// TIA Portal project "Ascensor" (V14)

(* hardware
DEVICE "S7-1200 station_1"  S7-1200 Station
   slot 0: "Rack_0"  S7-1200 Rack  Rack  V1.0
   slot 1: "PLC_1"  CPU 1214C AC/DC/Rly  6ES7 214-1BG40-0XB0  V4.0
*)

// ===== PLC "PLC_1"  CPU 1214C AC/DC/Rly =====

VAR_GLOBAL   // PLC tag table "Estados"
   "0" AT %M10.0 : Bool;   // Marcha/Paro del sistema
   "1" AT %M10.1 : Bool;   // Marcha/Paro del sistema
   "2" AT %M10.2 : Bool;   // Marcha/Paro del sistema
   "10" AT %M10.3 : Bool;   // Selección modo
   "11" AT %M10.4 : Bool;   // Selección modo
   "12" AT %M10.5 : Bool;   // Selección modo
   "20" AT %M10.6 : Bool;   // Movimiento de la cabina
   "21" AT %M10.7 : Bool;   // Movimiento de la cabina
   "22" AT %M11.0 : Bool;   // Movimiento de la cabina
   "23" AT %M11.1 : Bool;   // Movimiento de la cabina
   "24" AT %M11.2 : Bool;   // Movimiento de la cabina
   "25" AT %M11.3 : Bool;   // Movimiento de la cabina
   "30" AT %M11.4 : Bool;   // Apertura y Cierre de Puerta
   "31" AT %M11.5 : Bool;   // Apertura y Cierre de Puerta
   "32" AT %M11.6 : Bool;   // Apertura y Cierre de Puerta
   "33" AT %M11.7 : Bool;   // Apertura y Cierre de Puerta
   "34" AT %M12.0 : Bool;   // Apertura y Cierre de Puerta
   "35" AT %M12.1 : Bool;   // Apertura y Cierre de Puerta
   "40" AT %M12.2 : Bool;   // Reset llamda y memoria
   "41" AT %M12.3 : Bool;   // Reset llamda y memoria
   "42" AT %M12.4 : Bool;   // Reset llamda y memoria
   "43" AT %M12.5 : Bool;   // Reset llamda y memoria
   "50" AT %M12.6 : Bool;   // Órdenes automáticas de subida y bajada
   "51" AT %M12.7 : Bool;   // Órdenes automáticas de subida y bajada
   "52" AT %M13.0 : Bool;   // Órdenes automáticas de subida y bajada
   "60" AT %M13.1 : Bool;   // Órdenes manuales de subida y bajada
   "61" AT %M13.2 : Bool;   // Órdenes manuales de subida y bajada
   "62" AT %M13.3 : Bool;   // Órdenes manuales de subida y bajada
   "63" AT %M13.4 : Bool;   // Órdenes manuales de subida y bajada
   "64" AT %M13.5 : Bool;   // Órdenes manuales de subida y bajada
   "65" AT %M13.6 : Bool;   // Órdenes manuales de subida y bajada
   "66" AT %M13.7 : Bool;   // Órdenes manuales de subida y bajada
   "70" AT %M14.0 : Bool;   // Detección de errores
   "71" AT %M14.1 : Bool;   // Detección de errores
   "72" AT %M14.2 : Bool;   // Detección de errores
   "73" AT %M14.3 : Bool;   // Detección de errores
   "74" AT %M14.4 : Bool;   // Detección de errores
   "75" AT %M14.5 : Bool;   // Detección de errores
   "80" AT %M14.6 : Bool;   // Gestión de errores
   "81" AT %M14.7 : Bool;   // Gestión de errores
   "82" AT %M15.0 : Bool;   // Gestión de errores
   "83" AT %M15.1 : Bool;   // Gestión de errores
   "84" AT %M15.2 : Bool;   // Gestión de errores
   "85" AT %M15.3 : Bool;   // Gestión de errores
   "86" AT %M15.4 : Bool;   // Gestión de errores
   "87" AT %M15.5 : Bool;   // Gestión de errores
   "88" AT %M15.6 : Bool;   // Gestión de errores
   "90" AT %M15.7 : Bool;   // Descenso a primera planta
   "91" AT %M16.0 : Bool;   // Descenso a primera planta
   "92" AT %M16.1 : Bool;   // Descenso a primera planta
END_VAR

VAR_GLOBAL   // PLC tag table "Salidas"
   "LBC0" AT %M30.0 : Bool;   // Lámpara Pulsador Cabina Planta 0
   "LBC1" AT %M30.1 : Bool;   // Lámpara Pulsador Cabina Planta 1
   "LBC2" AT %M30.2 : Bool;   // Lámpara Pulsador Cabina Planta 2
   "LBC3" AT %M30.3 : Bool;   // Lámpara Pulsador Cabina Planta 3
   "LBP0" AT %M30.4 : Bool;   // Lámpara Pulsador Planta 0
   "LBP1" AT %M30.5 : Bool;   // Lámpara Pulsador Planta 1
   "LBP2" AT %M30.6 : Bool;   // Lámpara Pulsador Planta 2
   "LBP3" AT %M30.7 : Bool;   // Lámpara Pulsador Planta 3
   "MCD" AT %M31.0 : Bool;   // Orden Giro Motor Cabina Derecha - Ascender
   "MCI" AT %M31.1 : Bool;   // Orden Giro Motor Cabina Izquierda - Descender
   "MPD" AT %M31.2 : Bool;   // Orden Giro Motor Puerta Derecha - Apertura
   "MPI" AT %M31.3 : Bool;   // Orden Giro Motor Puerta Izquierda - Cierre
   "LA" AT %M31.4 : Bool;   // Lámpara Indicadora Llamada Ascendente
   "LD" AT %M31.5 : Bool;   // Lámpara Indicadora Llamada Descendente
   "Z" AT %M31.6 : Bool;   // Zumbador Indicador de Llamada
END_VAR

VAR_GLOBAL   // PLC tag table "Variables Internas"
   "Pos0" AT %M20.0 : Bool;   // Cabina en Planta 0
   "Pos1" AT %M20.1 : Bool;   // Cabina en Planta 1
   "Pos2" AT %M20.2 : Bool;   // Cabina en Planta 2
   "Pos3" AT %M20.3 : Bool;   // Cabina en Planta 3
   "Call0" AT %M20.4 : Bool;   // Llamada en Planta 0
   "Call1" AT %M20.5 : Bool;   // Llamada en Planta 1
   "Call2" AT %M20.6 : Bool;   // Llamada en Planta 2
   "Call3" AT %M20.7 : Bool;   // Llamada en Planta 3
   "hayCall" AT %M21.0 : Bool;   // Existencia Llamadas Pendietnes
   "upCall" AT %M21.1 : Bool;   // Llamada Ascender
   "downCall" AT %M21.2 : Bool;   // Llamada Descender
   "call_currentFloor" AT %M21.3 : Bool;   // Posición Cabina coincide con llamada
   "resetCall" AT %M21.4 : Bool;   // Finalizar llamda respondida
   "memUp" AT %M21.5 : Bool;   // Memoria Cabina Ascendiendo
   "memDown" AT %M21.6 : Bool;   // Memoria Cabina Descendiendo
   "sistemaActivado" AT %M21.7 : Bool;   // Estado General del Sistema
   "descenderPrimeraPlanta" AT %M22.0 : Bool;   // Descender a la primera planta
   "modoManual" AT %M22.1 : Bool;   // Activación del modo manual
   "modoAuto" AT %M22.2 : Bool;   // Activación del modo automático
   "abrirPuertas" AT %M22.3 : Bool;   // Iniciar secuencia de apertura de puertas
   "esperandoOrden" AT %M22.4 : Bool;   // Iniciar secuencia de decisión sobre el movimiento
   "error1" AT %M22.5 : Bool;   // Indicador de emergencia tipo 1
   "error2" AT %M22.6 : Bool;   // Indicador de emergencia tipo 2
   "modoSeguridad" AT %M22.7 : Bool;   // Indicador del estado del sistema
   "moveUp" AT %M23.0 : Bool;   // Orden de ascender
   "moveDown" AT %M23.1 : Bool;   // Orden de descender
   "finalizaLlamada" AT %M23.2 : Bool;   // Resetea una llamada
   "deleteAllCalls" AT %M23.3 : Bool;   // Resetea todas las llamadas
END_VAR

VAR_GLOBAL   // PLC tag table "Entradas"
   "BC0" AT %M0.0 : Bool;   // Pulsador Cabina Planta 0
   "BC1" AT %M0.1 : Bool;   // Pulsador Cabina Planta 1
   "BC2" AT %M0.2 : Bool;   // Pulsador Cabina Planta 2
   "BC3" AT %M0.3 : Bool;   // Pulsador Cabina Planta 3
   "BCC" AT %M0.4 : Bool;   // Pulsador Cabina Cierre Puertas
   "BCA" AT %M0.5 : Bool;   // Pulsador Cabina Apertura Puertas
   "BP0" AT %M0.6 : Bool;   // Pulsador Planta 0
   "BP1" AT %M0.7 : Bool;   // Pulsador Planta 1
   "BP2" AT %M1.0 : Bool;   // Pulsador Planta 2
   "BP3" AT %M1.1 : Bool;   // Pulsador Planta 3
   "IBL0" AT %M1.2 : Bool;   // Interruptor Biestable Lengüeta Planta 0
   "IBL1" AT %M1.3 : Bool;   // Interruptor Biestable Lengüeta Planta 1
   "IBL2" AT %M1.4 : Bool;   // Interruptor Biestable Lengüeta Planta 2
   "IBL3" AT %M1.5 : Bool;   // Interruptor Biestable Lengüeta Planta 3
   "FCPA" AT %M1.6 : Bool;   // Final de Carrera Puerta Apertura
   "FCPC" AT %M1.7 : Bool;   // Final de Carrera Puerta Cierre
   "SO" AT %M2.0 : Bool;   // Sensor Obstáculo Puerta Cabina
   "SC" AT %M2.1 : Bool;   // Sensor Carga Cabina
   "Activar" AT %M2.2 : Bool;   // Señal de Activación del sistema
   "Desactivar" AT %M2.3 : Bool;   // Señal de Desactivación del sistema
   "MA" AT %M2.4 : Bool;   // Señal de selección del modo manual
   "AUTO" AT %M2.5 : Bool;   // Señal de selección del modo automático
   "emergenciaParada" AT %M2.6 : Bool;   // Señal de emergencia que requiere parada
   "finEmergenciaParada" AT %M2.7 : Bool;   // Señal fin de emergencia que requiere parada
   "emergenciaPrimeraPlanta" AT %M3.0 : Bool;   // Señal de emergencia que requiere descender a la primera planta
   "finEmergenciaPrimeraPlanta" AT %M3.1 : Bool;   // Señal de fin de emergencia que requiere descender a primera planta
   "BA" AT %M3.2 : Bool;   // Botón Ascender Manual
   "BD" AT %M3.3 : Bool;   // Botón Descender Manual
   "BI" AT %M3.4 : Bool;   // Botón Ignorar Manual
END_VAR

// folder: System blocks/Program resources

DATA_BLOCK "TimerPuertas"   // DB3
{ S7_Optimized_Access := 'TRUE' }
AUTHOR : Simatic
FAMILY : IEC
NAME : IEC_TMR
VERSION : 1.0
// stored: InstanceOfName IEC_TIMER
"IEC_TIMER"
BEGIN
END_DATA_BLOCK

// folder: (top level)

ORGANIZATION_BLOCK "Main"   // OB1, LAD, ProgramCycle
TITLE = "Main Program Sweep (Cycle)"
{ S7_Optimized_Access := 'TRUE' }
VERSION : 0.1
   VAR_INPUT
      Initial_Call : Bool;   // Initial call of this OB
      Remanence : Bool;   // =True, if remanent data are available
   END_VAR
   VAR_TEMP   // added for the SCL form of the ladder/FBD networks
      _w1 : Bool;
      _w2 : Bool;
      _w3 : Bool;
   END_VAR
BEGIN

REGION Network 1: Variables Internas Posición Cabina
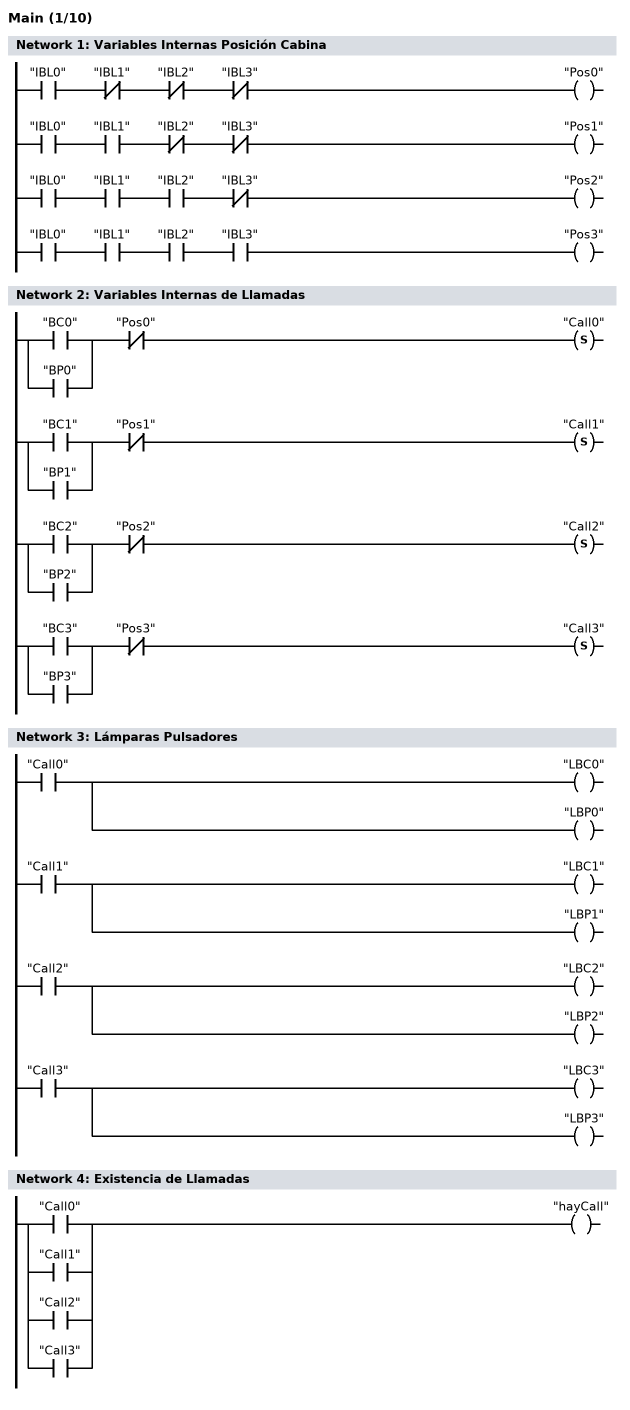
   RUNG wire#powerrail
      Contact( "IBL0" )
      I_Contact( "IBL1" )
      I_Contact( "IBL2" )
      I_Contact( "IBL3" )
      Coil( "Pos0" )
   END_RUNG
   RUNG wire#powerrail
      Contact( "IBL0" )
      Contact( "IBL1" )
      I_Contact( "IBL2" )
      I_Contact( "IBL3" )
      Coil( "Pos1" )
   END_RUNG
   RUNG wire#powerrail
      Contact( "IBL0" )
      Contact( "IBL1" )
      Contact( "IBL2" )
      I_Contact( "IBL3" )
      Coil( "Pos2" )
   END_RUNG
   RUNG wire#powerrail
      Contact( "IBL0" )
      Contact( "IBL1" )
      Contact( "IBL2" )
      Contact( "IBL3" )
      Coil( "Pos3" )
   END_RUNG
   // the same network as SCL:
   "Pos0" := "IBL0" AND NOT "IBL1" AND NOT "IBL2" AND NOT "IBL3";
   "Pos1" := "IBL0" AND "IBL1" AND NOT "IBL2" AND NOT "IBL3";
   "Pos2" := "IBL0" AND "IBL1" AND "IBL2" AND NOT "IBL3";
   "Pos3" := "IBL0" AND "IBL1" AND "IBL2" AND "IBL3";
END_REGION

REGION Network 2: Variables Internas de Llamadas
   RUNG wire#powerrail
      Contact( "BC0" )
      wire#w1
      I_Contact( "Pos0" )
      S_Coil( "Call0" )
   END_RUNG
   RUNG wire#powerrail
      Contact( "BP0" )
   END_RUNG wire#w1
   RUNG wire#powerrail
      Contact( "BC1" )
      wire#w2
      I_Contact( "Pos1" )
      S_Coil( "Call1" )
   END_RUNG
   RUNG wire#powerrail
      Contact( "BP1" )
   END_RUNG wire#w2
   RUNG wire#powerrail
      Contact( "BC2" )
      wire#w3
      I_Contact( "Pos2" )
      S_Coil( "Call2" )
   END_RUNG
   RUNG wire#powerrail
      Contact( "BP2" )
   END_RUNG wire#w3
   RUNG wire#powerrail
      Contact( "BC3" )
      wire#w4
      I_Contact( "Pos3" )
      S_Coil( "Call3" )
   END_RUNG
   RUNG wire#powerrail
      Contact( "BP3" )
   END_RUNG wire#w4
   // the same network as SCL:
   IF ("BC0" OR "BP0") AND NOT "Pos0" THEN "Call0" := TRUE; END_IF;
   IF ("BC1" OR "BP1") AND NOT "Pos1" THEN "Call1" := TRUE; END_IF;
   IF ("BC2" OR "BP2") AND NOT "Pos2" THEN "Call2" := TRUE; END_IF;
   IF ("BC3" OR "BP3") AND NOT "Pos3" THEN "Call3" := TRUE; END_IF;
END_REGION

REGION Network 3: Lámparas Pulsadores
   RUNG wire#powerrail
      Contact( "Call0" )
      wire#w1
      Coil( "LBC0" )
   END_RUNG
   RUNG wire#w1
      Coil( "LBP0" )
   END_RUNG
   RUNG wire#powerrail
      Contact( "Call1" )
      wire#w2
      Coil( "LBC1" )
   END_RUNG
   RUNG wire#w2
      Coil( "LBP1" )
   END_RUNG
   RUNG wire#powerrail
      Contact( "Call2" )
      wire#w3
      Coil( "LBC2" )
   END_RUNG
   RUNG wire#w3
      Coil( "LBP2" )
   END_RUNG
   RUNG wire#powerrail
      Contact( "Call3" )
      wire#w4
      Coil( "LBC3" )
   END_RUNG
   RUNG wire#w4
      Coil( "LBP3" )
   END_RUNG
   // the same network as SCL:
   "LBC0" := "Call0";
   "LBP0" := "Call0";
   "LBC1" := "Call1";
   "LBP1" := "Call1";
   "LBC2" := "Call2";
   "LBP2" := "Call2";
   "LBC3" := "Call3";
   "LBP3" := "Call3";
END_REGION

REGION Network 4: Existencia de Llamadas
   RUNG wire#powerrail
      Contact( "Call0" )
      wire#w1
      Coil( "hayCall" )
   END_RUNG
   RUNG wire#powerrail
      Contact( "Call1" )
   END_RUNG wire#w1
   RUNG wire#powerrail
      Contact( "Call2" )
   END_RUNG wire#w1
   RUNG wire#powerrail
      Contact( "Call3" )
   END_RUNG wire#w1
   // the same network as SCL:
   "hayCall" := "Call0" OR "Call1" OR "Call2" OR "Call3";
END_REGION

REGION Network 5: Dirección de las llamadas
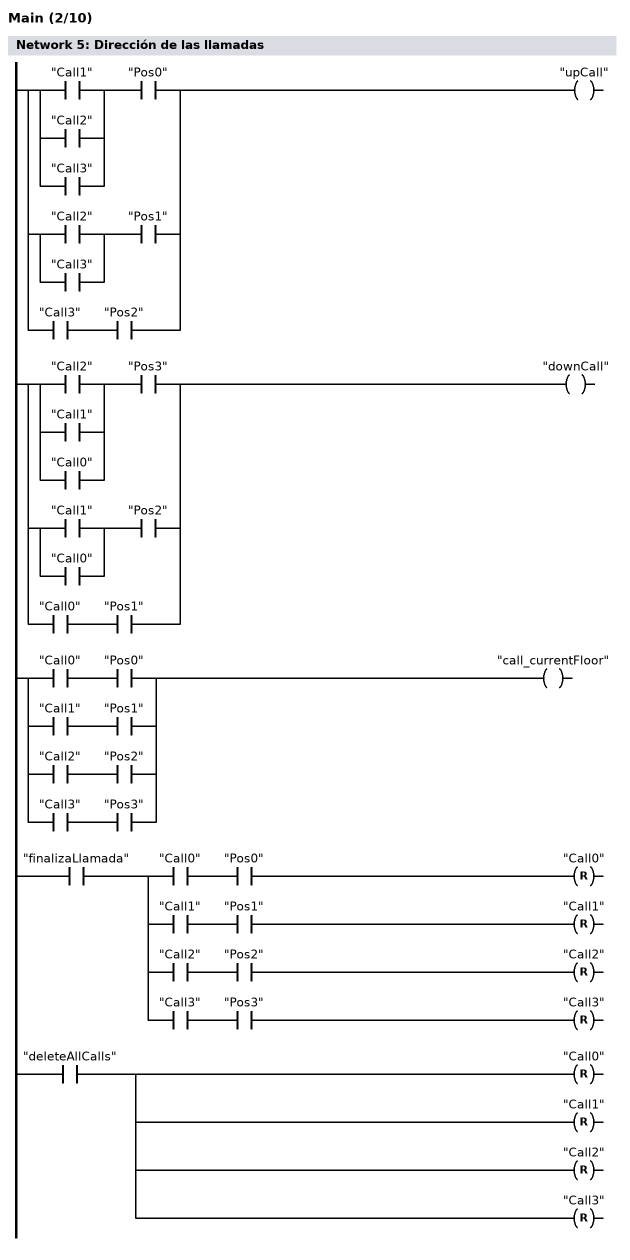
   RUNG wire#powerrail
      Contact( "Call1" )
      wire#w1
      Contact( "Pos0" )
      wire#w2
      Coil( "upCall" )
   END_RUNG
   RUNG wire#powerrail
      Contact( "Call2" )
   END_RUNG wire#w1
   RUNG wire#powerrail
      Contact( "Call3" )
   END_RUNG wire#w1
   RUNG wire#powerrail
      Contact( "Call2" )
      wire#w3
      Contact( "Pos1" )
   END_RUNG wire#w2
   RUNG wire#powerrail
      Contact( "Call3" )
   END_RUNG wire#w3
   RUNG wire#powerrail
      Contact( "Call3" )
      Contact( "Pos2" )
   END_RUNG wire#w2
   RUNG wire#powerrail
      Contact( "Call2" )
      wire#w4
      Contact( "Pos3" )
      wire#w5
      Coil( "downCall" )
   END_RUNG
   RUNG wire#powerrail
      Contact( "Call1" )
   END_RUNG wire#w4
   RUNG wire#powerrail
      Contact( "Call0" )
   END_RUNG wire#w4
   RUNG wire#powerrail
      Contact( "Call1" )
      wire#w6
      Contact( "Pos2" )
   END_RUNG wire#w5
   RUNG wire#powerrail
      Contact( "Call0" )
   END_RUNG wire#w6
   RUNG wire#powerrail
      Contact( "Call0" )
      Contact( "Pos1" )
   END_RUNG wire#w5
   RUNG wire#powerrail
      Contact( "Call0" )
      Contact( "Pos0" )
      wire#w7
      Coil( "call_currentFloor" )
   END_RUNG
   RUNG wire#powerrail
      Contact( "Call1" )
      Contact( "Pos1" )
   END_RUNG wire#w7
   RUNG wire#powerrail
      Contact( "Call2" )
      Contact( "Pos2" )
   END_RUNG wire#w7
   RUNG wire#powerrail
      Contact( "Call3" )
      Contact( "Pos3" )
   END_RUNG wire#w7
   RUNG wire#powerrail
      Contact( "finalizaLlamada" )
      wire#w8
      Contact( "Call0" )
      Contact( "Pos0" )
      R_Coil( "Call0" )
   END_RUNG
   RUNG wire#w8
      Contact( "Call1" )
      Contact( "Pos1" )
      R_Coil( "Call1" )
   END_RUNG
   RUNG wire#w8
      Contact( "Call2" )
      Contact( "Pos2" )
      R_Coil( "Call2" )
   END_RUNG
   RUNG wire#w8
      Contact( "Call3" )
      Contact( "Pos3" )
      R_Coil( "Call3" )
   END_RUNG
   RUNG wire#powerrail
      Contact( "deleteAllCalls" )
      wire#w9
      R_Coil( "Call0" )
   END_RUNG
   RUNG wire#w9
      R_Coil( "Call1" )
   END_RUNG
   RUNG wire#w9
      R_Coil( "Call2" )
   END_RUNG
   RUNG wire#w9
      R_Coil( "Call3" )
   END_RUNG
   // the same network as SCL:
   "upCall" := (("Call1" OR "Call2" OR "Call3") AND "Pos0") OR (("Call2" OR "Call3") AND "Pos1") OR ("Call3" AND "Pos2");
   "downCall" := (("Call2" OR "Call1" OR "Call0") AND "Pos3") OR (("Call1" OR "Call0") AND "Pos2") OR ("Call0" AND "Pos1");
   "call_currentFloor" := ("Call0" AND "Pos0") OR ("Call1" AND "Pos1") OR ("Call2" AND "Pos2") OR ("Call3" AND "Pos3");
   IF "finalizaLlamada" AND "Call0" AND "Pos0" THEN "Call0" := FALSE; END_IF;
   IF "finalizaLlamada" AND "Call1" AND "Pos1" THEN "Call1" := FALSE; END_IF;
   IF "finalizaLlamada" AND "Call2" AND "Pos2" THEN "Call2" := FALSE; END_IF;
   IF "finalizaLlamada" AND "Call3" AND "Pos3" THEN "Call3" := FALSE; END_IF;
   IF "deleteAllCalls" THEN
       "Call0" := FALSE;
       "Call1" := FALSE;
       "Call2" := FALSE;
       "Call3" := FALSE;
   END_IF;
END_REGION

REGION Network 6: Marcha/Paro del sistema
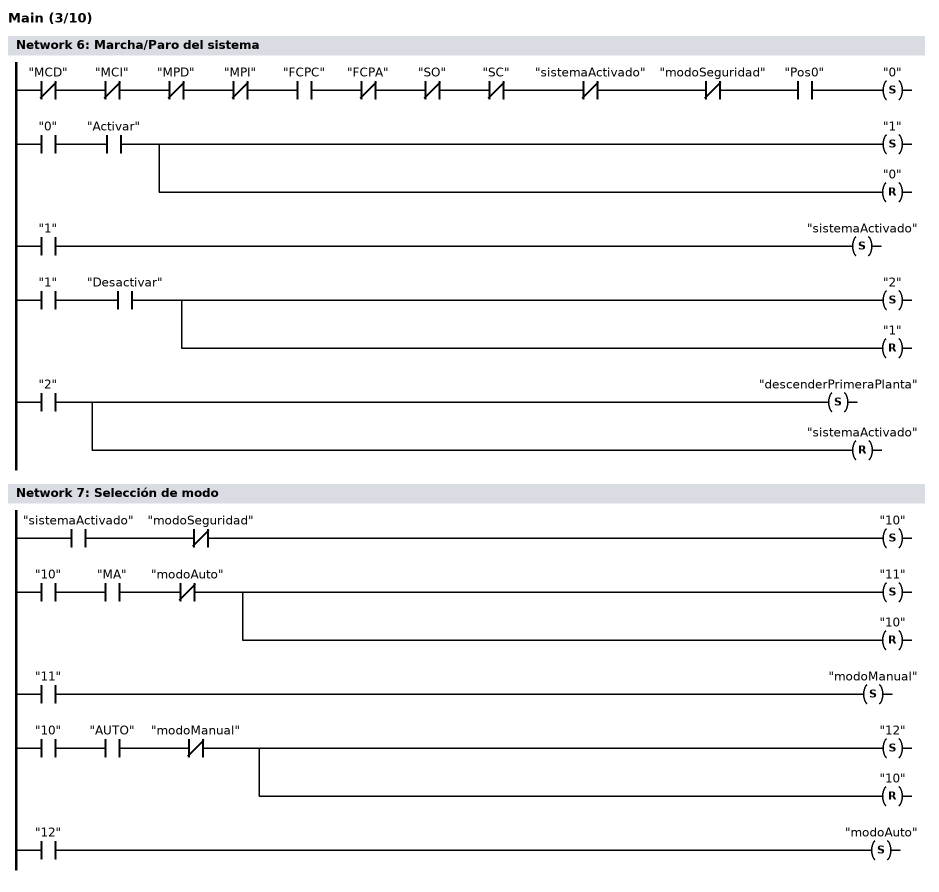
   RUNG wire#powerrail
      I_Contact( "MCD" )
      I_Contact( "MCI" )
      I_Contact( "MPD" )
      I_Contact( "MPI" )
      Contact( "FCPC" )
      I_Contact( "FCPA" )
      I_Contact( "SO" )
      I_Contact( "SC" )
      I_Contact( "sistemaActivado" )
      I_Contact( "modoSeguridad" )
      Contact( "Pos0" )
      S_Coil( "0" )
   END_RUNG
   RUNG wire#powerrail
      Contact( "0" )
      Contact( "Activar" )
      wire#w1
      S_Coil( "1" )
   END_RUNG
   RUNG wire#w1
      R_Coil( "0" )
   END_RUNG
   RUNG wire#powerrail
      Contact( "1" )
      S_Coil( "sistemaActivado" )
   END_RUNG
   RUNG wire#powerrail
      Contact( "1" )
      Contact( "Desactivar" )
      wire#w2
      S_Coil( "2" )
   END_RUNG
   RUNG wire#w2
      R_Coil( "1" )
   END_RUNG
   RUNG wire#powerrail
      Contact( "2" )
      wire#w3
      S_Coil( "descenderPrimeraPlanta" )
   END_RUNG
   RUNG wire#w3
      R_Coil( "sistemaActivado" )
   END_RUNG
   // the same network as SCL:
   IF NOT "MCD" AND NOT "MCI" AND NOT "MPD" AND NOT "MPI" AND "FCPC" AND NOT "FCPA" AND NOT "SO" AND NOT "SC" AND NOT "sistemaActivado" AND NOT "modoSeguridad" AND "Pos0" THEN
       "0" := TRUE;
   END_IF;
   IF "0" AND "Activar" THEN
       "1" := TRUE;
       "0" := FALSE;
   END_IF;
   IF "1" THEN "sistemaActivado" := TRUE; END_IF;
   IF "1" AND "Desactivar" THEN
       "2" := TRUE;
       "1" := FALSE;
   END_IF;
   IF "2" THEN
       "descenderPrimeraPlanta" := TRUE;
       "sistemaActivado" := FALSE;
   END_IF;
END_REGION

REGION Network 7: Selección de modo
   RUNG wire#powerrail
      Contact( "sistemaActivado" )
      I_Contact( "modoSeguridad" )
      S_Coil( "10" )
   END_RUNG
   RUNG wire#powerrail
      Contact( "10" )
      Contact( "MA" )
      I_Contact( "modoAuto" )
      wire#w1
      S_Coil( "11" )
   END_RUNG
   RUNG wire#w1
      R_Coil( "10" )
   END_RUNG
   RUNG wire#powerrail
      Contact( "11" )
      S_Coil( "modoManual" )
   END_RUNG
   RUNG wire#powerrail
      Contact( "10" )
      Contact( "AUTO" )
      I_Contact( "modoManual" )
      wire#w2
      S_Coil( "12" )
   END_RUNG
   RUNG wire#w2
      R_Coil( "10" )
   END_RUNG
   RUNG wire#powerrail
      Contact( "12" )
      S_Coil( "modoAuto" )
   END_RUNG
   // the same network as SCL:
   IF "sistemaActivado" AND NOT "modoSeguridad" THEN "10" := TRUE; END_IF;
   IF "10" AND "MA" AND NOT "modoAuto" THEN
       "11" := TRUE;
       "10" := FALSE;
   END_IF;
   IF "11" THEN "modoManual" := TRUE; END_IF;
   IF "10" AND "AUTO" AND NOT "modoManual" THEN
       "12" := TRUE;
       "10" := FALSE;
   END_IF;
   IF "12" THEN "modoAuto" := TRUE; END_IF;
END_REGION

REGION Network 8: Movimiento de la cabina
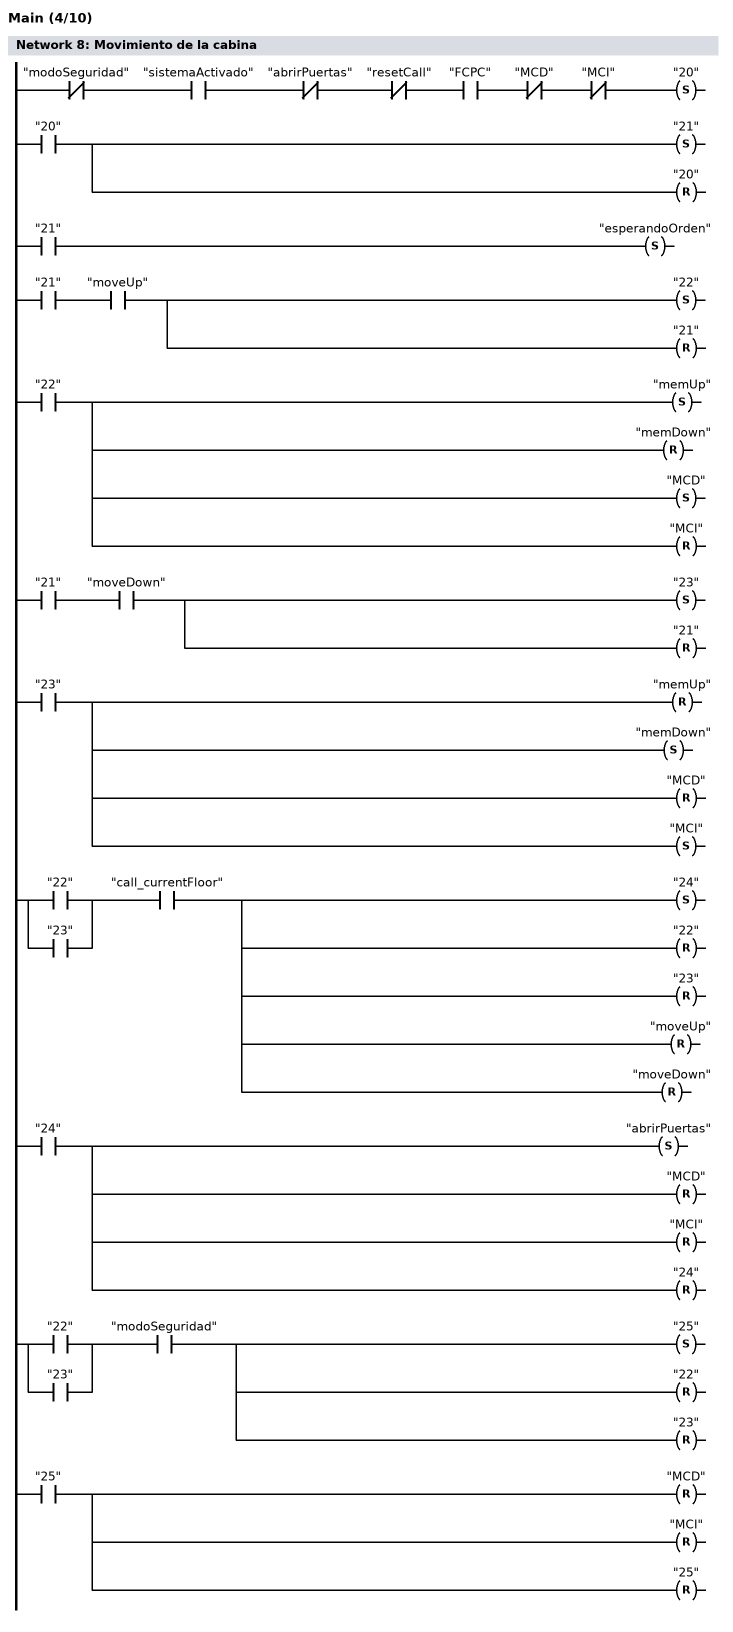
   RUNG wire#powerrail
      I_Contact( "modoSeguridad" )
      Contact( "sistemaActivado" )
      I_Contact( "abrirPuertas" )
      I_Contact( "resetCall" )
      Contact( "FCPC" )
      I_Contact( "MCD" )
      I_Contact( "MCI" )
      S_Coil( "20" )
   END_RUNG
   RUNG wire#powerrail
      Contact( "20" )
      wire#w1
      S_Coil( "21" )
   END_RUNG
   RUNG wire#w1
      R_Coil( "20" )
   END_RUNG
   RUNG wire#powerrail
      Contact( "21" )
      S_Coil( "esperandoOrden" )
   END_RUNG
   RUNG wire#powerrail
      Contact( "21" )
      Contact( "moveUp" )
      wire#w2
      S_Coil( "22" )
   END_RUNG
   RUNG wire#w2
      R_Coil( "21" )
   END_RUNG
   RUNG wire#powerrail
      Contact( "22" )
      wire#w3
      S_Coil( "memUp" )
   END_RUNG
   RUNG wire#w3
      R_Coil( "memDown" )
   END_RUNG
   RUNG wire#w3
      S_Coil( "MCD" )
   END_RUNG
   RUNG wire#w3
      R_Coil( "MCI" )
   END_RUNG
   RUNG wire#powerrail
      Contact( "21" )
      Contact( "moveDown" )
      wire#w4
      S_Coil( "23" )
   END_RUNG
   RUNG wire#w4
      R_Coil( "21" )
   END_RUNG
   RUNG wire#powerrail
      Contact( "23" )
      wire#w5
      R_Coil( "memUp" )
   END_RUNG
   RUNG wire#w5
      S_Coil( "memDown" )
   END_RUNG
   RUNG wire#w5
      R_Coil( "MCD" )
   END_RUNG
   RUNG wire#w5
      S_Coil( "MCI" )
   END_RUNG
   RUNG wire#powerrail
      Contact( "22" )
      wire#w6
      Contact( "call_currentFloor" )
      wire#w7
      S_Coil( "24" )
   END_RUNG
   RUNG wire#powerrail
      Contact( "23" )
   END_RUNG wire#w6
   RUNG wire#w7
      R_Coil( "22" )
   END_RUNG
   RUNG wire#w7
      R_Coil( "23" )
   END_RUNG
   RUNG wire#w7
      R_Coil( "moveUp" )
   END_RUNG
   RUNG wire#w7
      R_Coil( "moveDown" )
   END_RUNG
   RUNG wire#powerrail
      Contact( "24" )
      wire#w8
      S_Coil( "abrirPuertas" )
   END_RUNG
   RUNG wire#w8
      R_Coil( "MCD" )
   END_RUNG
   RUNG wire#w8
      R_Coil( "MCI" )
   END_RUNG
   RUNG wire#w8
      R_Coil( "24" )
   END_RUNG
   RUNG wire#powerrail
      Contact( "22" )
      wire#w9
      Contact( "modoSeguridad" )
      wire#w10
      S_Coil( "25" )
   END_RUNG
   RUNG wire#powerrail
      Contact( "23" )
   END_RUNG wire#w9
   RUNG wire#w10
      R_Coil( "22" )
   END_RUNG
   RUNG wire#w10
      R_Coil( "23" )
   END_RUNG
   RUNG wire#powerrail
      Contact( "25" )
      wire#w11
      R_Coil( "MCD" )
   END_RUNG
   RUNG wire#w11
      R_Coil( "MCI" )
   END_RUNG
   RUNG wire#w11
      R_Coil( "25" )
   END_RUNG
   // the same network as SCL:
   IF NOT "modoSeguridad" AND "sistemaActivado" AND NOT "abrirPuertas" AND NOT "resetCall" AND "FCPC" AND NOT "MCD" AND NOT "MCI" THEN
       "20" := TRUE;
   END_IF;
   IF "20" THEN
       "21" := TRUE;
       "20" := FALSE;
   END_IF;
   IF "21" THEN "esperandoOrden" := TRUE; END_IF;
   IF "21" AND "moveUp" THEN
       "22" := TRUE;
       "21" := FALSE;
   END_IF;
   IF "22" THEN
       "memUp" := TRUE;
       "memDown" := FALSE;
       "MCD" := TRUE;
       "MCI" := FALSE;
   END_IF;
   IF "21" AND "moveDown" THEN
       "23" := TRUE;
       "21" := FALSE;
   END_IF;
   IF "23" THEN
       "memUp" := FALSE;
       "memDown" := TRUE;
       "MCD" := FALSE;
       "MCI" := TRUE;
   END_IF;
   IF ("22" OR "23") AND "call_currentFloor" THEN "24" := TRUE; END_IF;
   #_w1 := ("22" OR "23") AND "call_currentFloor";
   IF #_w1 THEN
       "22" := FALSE;
       "23" := FALSE;
       "moveUp" := FALSE;
       "moveDown" := FALSE;
   END_IF;
   IF "24" THEN
       "abrirPuertas" := TRUE;
       "MCD" := FALSE;
       "MCI" := FALSE;
       "24" := FALSE;
   END_IF;
   IF ("22" OR "23") AND "modoSeguridad" THEN "25" := TRUE; END_IF;
   #_w2 := ("22" OR "23") AND "modoSeguridad";
   IF #_w2 THEN
       "22" := FALSE;
       "23" := FALSE;
   END_IF;
   IF "25" THEN
       "MCD" := FALSE;
       "MCI" := FALSE;
       "25" := FALSE;
   END_IF;
END_REGION

REGION Network 9: Apertura y cierre de puertas
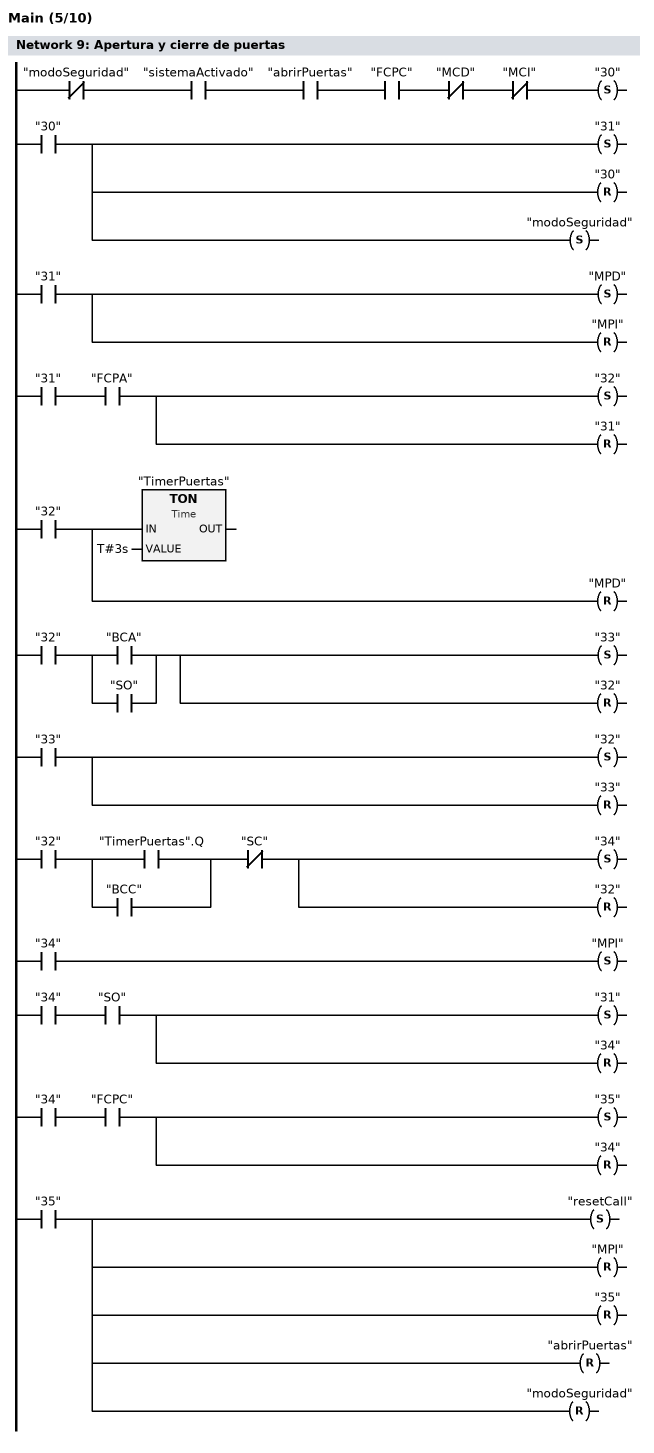
   IF NOT "modoSeguridad" AND "sistemaActivado" AND "abrirPuertas" AND "FCPC" AND NOT "MCD" AND NOT "MCI" THEN
       "30" := TRUE;
   END_IF;
   IF "30" THEN "31" := TRUE; END_IF;
   #_w1 := "30";
   IF #_w1 THEN
       "30" := FALSE;
       "modoSeguridad" := TRUE;
   END_IF;
   IF "31" THEN
       "MPD" := TRUE;
       "MPI" := FALSE;
   END_IF;
   IF "31" AND "FCPA" THEN
       "32" := TRUE;
       "31" := FALSE;
   END_IF;
   "TimerPuertas".TON(IN := "32", PT := T#3s);   // TON coil
   IF "32" THEN "MPD" := FALSE; END_IF;
   IF "32" AND ("BCA" OR "SO") THEN
       "33" := TRUE;
       "32" := FALSE;
   END_IF;
   IF "33" THEN
       "32" := TRUE;
       "33" := FALSE;
   END_IF;
   IF "32" AND ("TimerPuertas".Q OR "BCC") AND NOT "SC" THEN
       "34" := TRUE;
       "32" := FALSE;
   END_IF;
   IF "34" THEN "MPI" := TRUE; END_IF;
   IF "34" AND "SO" THEN
       "31" := TRUE;
       "34" := FALSE;
   END_IF;
   IF "34" AND "FCPC" THEN
       "35" := TRUE;
       "34" := FALSE;
   END_IF;
   IF "35" THEN
       "resetCall" := TRUE;
       "MPI" := FALSE;
   END_IF;
   #_w2 := "35";
   IF #_w2 THEN
       "35" := FALSE;
       "abrirPuertas" := FALSE;
       "modoSeguridad" := FALSE;
   END_IF;
END_REGION

REGION Network 10: Reset de llamada y memoria
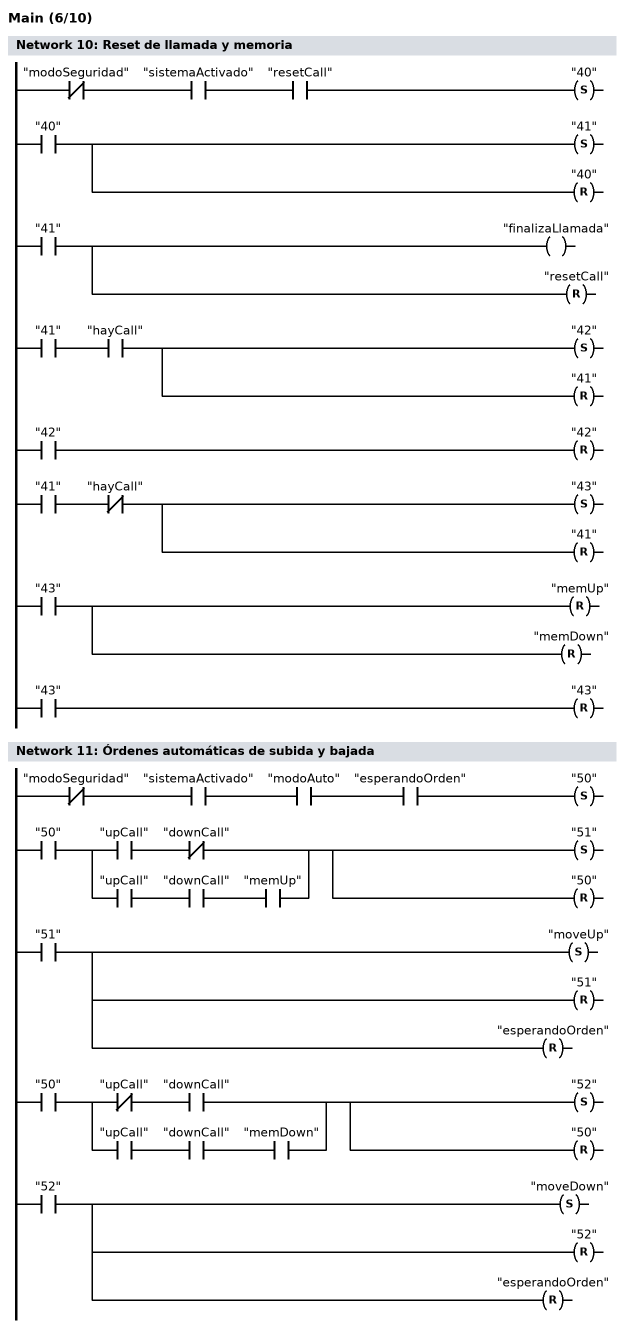
   RUNG wire#powerrail
      I_Contact( "modoSeguridad" )
      Contact( "sistemaActivado" )
      Contact( "resetCall" )
      S_Coil( "40" )
   END_RUNG
   RUNG wire#powerrail
      Contact( "40" )
      wire#w1
      S_Coil( "41" )
   END_RUNG
   RUNG wire#w1
      R_Coil( "40" )
   END_RUNG
   RUNG wire#powerrail
      Contact( "41" )
      wire#w2
      Coil( "finalizaLlamada" )
   END_RUNG
   RUNG wire#w2
      R_Coil( "resetCall" )
   END_RUNG
   RUNG wire#powerrail
      Contact( "41" )
      Contact( "hayCall" )
      wire#w3
      S_Coil( "42" )
   END_RUNG
   RUNG wire#w3
      R_Coil( "41" )
   END_RUNG
   RUNG wire#powerrail
      Contact( "42" )
      R_Coil( "42" )
   END_RUNG
   RUNG wire#powerrail
      Contact( "41" )
      I_Contact( "hayCall" )
      wire#w4
      S_Coil( "43" )
   END_RUNG
   RUNG wire#w4
      R_Coil( "41" )
   END_RUNG
   RUNG wire#powerrail
      Contact( "43" )
      wire#w5
      R_Coil( "memUp" )
   END_RUNG
   RUNG wire#w5
      R_Coil( "memDown" )
   END_RUNG
   RUNG wire#powerrail
      Contact( "43" )
      R_Coil( "43" )
   END_RUNG
   // the same network as SCL:
   IF NOT "modoSeguridad" AND "sistemaActivado" AND "resetCall" THEN "40" := TRUE; END_IF;
   IF "40" THEN
       "41" := TRUE;
       "40" := FALSE;
   END_IF;
   "finalizaLlamada" := "41";
   IF "41" THEN "resetCall" := FALSE; END_IF;
   IF "41" AND "hayCall" THEN
       "42" := TRUE;
       "41" := FALSE;
   END_IF;
   IF "42" THEN "42" := FALSE; END_IF;
   IF "41" AND NOT "hayCall" THEN
       "43" := TRUE;
       "41" := FALSE;
   END_IF;
   IF "43" THEN
       "memUp" := FALSE;
       "memDown" := FALSE;
       "43" := FALSE;
   END_IF;
END_REGION

REGION Network 11: Órdenes automáticas de subida y bajada
   RUNG wire#powerrail
      I_Contact( "modoSeguridad" )
      Contact( "sistemaActivado" )
      Contact( "modoAuto" )
      Contact( "esperandoOrden" )
      S_Coil( "50" )
   END_RUNG
   RUNG wire#powerrail
      Contact( "50" )
      wire#w1
      Contact( "upCall" )
      I_Contact( "downCall" )
      wire#w2
      S_Coil( "51" )
   END_RUNG
   RUNG wire#w1
      Contact( "upCall" )
      Contact( "downCall" )
      Contact( "memUp" )
   END_RUNG wire#w2
   RUNG wire#w2
      R_Coil( "50" )
   END_RUNG
   RUNG wire#powerrail
      Contact( "51" )
      wire#w3
      S_Coil( "moveUp" )
   END_RUNG
   RUNG wire#w3
      R_Coil( "51" )
   END_RUNG
   RUNG wire#w3
      R_Coil( "esperandoOrden" )
   END_RUNG
   RUNG wire#powerrail
      Contact( "50" )
      wire#w4
      I_Contact( "upCall" )
      Contact( "downCall" )
      wire#w5
      S_Coil( "52" )
   END_RUNG
   RUNG wire#w4
      Contact( "upCall" )
      Contact( "downCall" )
      Contact( "memDown" )
   END_RUNG wire#w5
   RUNG wire#w5
      R_Coil( "50" )
   END_RUNG
   RUNG wire#powerrail
      Contact( "52" )
      wire#w6
      S_Coil( "moveDown" )
   END_RUNG
   RUNG wire#w6
      R_Coil( "52" )
   END_RUNG
   RUNG wire#w6
      R_Coil( "esperandoOrden" )
   END_RUNG
   // the same network as SCL:
   IF NOT "modoSeguridad" AND "sistemaActivado" AND "modoAuto" AND "esperandoOrden" THEN
       "50" := TRUE;
   END_IF;
   IF "50" AND (("upCall" AND NOT "downCall") OR ("upCall" AND "downCall" AND "memUp")) THEN
       "51" := TRUE;
       "50" := FALSE;
   END_IF;
   IF "51" THEN "moveUp" := TRUE; END_IF;
   #_w1 := "51";
   IF #_w1 THEN
       "51" := FALSE;
       "esperandoOrden" := FALSE;
   END_IF;
   IF "50" AND ((NOT "upCall" AND "downCall") OR ("upCall" AND "downCall" AND "memDown")) THEN
       "52" := TRUE;
       "50" := FALSE;
   END_IF;
   IF "52" THEN "moveDown" := TRUE; END_IF;
   #_w2 := "52";
   IF #_w2 THEN
       "52" := FALSE;
       "esperandoOrden" := FALSE;
   END_IF;
END_REGION

REGION Network 12: Órdenes manuales de subida y bajada
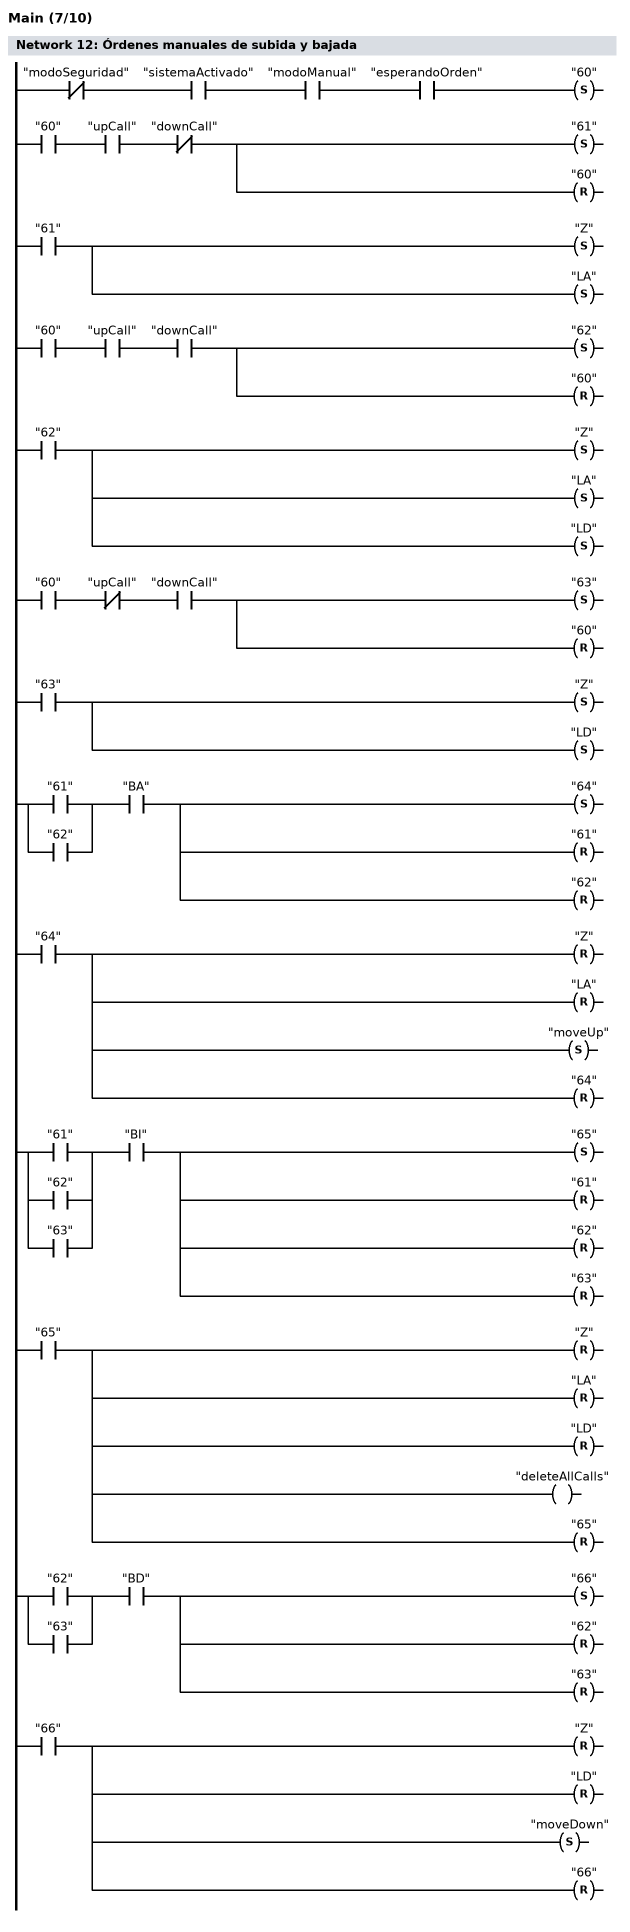
   RUNG wire#powerrail
      I_Contact( "modoSeguridad" )
      Contact( "sistemaActivado" )
      Contact( "modoManual" )
      Contact( "esperandoOrden" )
      S_Coil( "60" )
   END_RUNG
   RUNG wire#powerrail
      Contact( "60" )
      Contact( "upCall" )
      I_Contact( "downCall" )
      wire#w1
      S_Coil( "61" )
   END_RUNG
   RUNG wire#w1
      R_Coil( "60" )
   END_RUNG
   RUNG wire#powerrail
      Contact( "61" )
      wire#w2
      S_Coil( "Z" )
   END_RUNG
   RUNG wire#w2
      S_Coil( "LA" )
   END_RUNG
   RUNG wire#powerrail
      Contact( "60" )
      Contact( "upCall" )
      Contact( "downCall" )
      wire#w3
      S_Coil( "62" )
   END_RUNG
   RUNG wire#w3
      R_Coil( "60" )
   END_RUNG
   RUNG wire#powerrail
      Contact( "62" )
      wire#w4
      S_Coil( "Z" )
   END_RUNG
   RUNG wire#w4
      S_Coil( "LA" )
   END_RUNG
   RUNG wire#w4
      S_Coil( "LD" )
   END_RUNG
   RUNG wire#powerrail
      Contact( "60" )
      I_Contact( "upCall" )
      Contact( "downCall" )
      wire#w5
      S_Coil( "63" )
   END_RUNG
   RUNG wire#w5
      R_Coil( "60" )
   END_RUNG
   RUNG wire#powerrail
      Contact( "63" )
      wire#w6
      S_Coil( "Z" )
   END_RUNG
   RUNG wire#w6
      S_Coil( "LD" )
   END_RUNG
   RUNG wire#powerrail
      Contact( "61" )
      wire#w7
      Contact( "BA" )
      wire#w8
      S_Coil( "64" )
   END_RUNG
   RUNG wire#powerrail
      Contact( "62" )
   END_RUNG wire#w7
   RUNG wire#w8
      R_Coil( "61" )
   END_RUNG
   RUNG wire#w8
      R_Coil( "62" )
   END_RUNG
   RUNG wire#powerrail
      Contact( "64" )
      wire#w9
      R_Coil( "Z" )
   END_RUNG
   RUNG wire#w9
      R_Coil( "LA" )
   END_RUNG
   RUNG wire#w9
      S_Coil( "moveUp" )
   END_RUNG
   RUNG wire#w9
      R_Coil( "64" )
   END_RUNG
   RUNG wire#powerrail
      Contact( "61" )
      wire#w10
      Contact( "BI" )
      wire#w11
      S_Coil( "65" )
   END_RUNG
   RUNG wire#powerrail
      Contact( "62" )
   END_RUNG wire#w10
   RUNG wire#powerrail
      Contact( "63" )
   END_RUNG wire#w10
   RUNG wire#w11
      R_Coil( "61" )
   END_RUNG
   RUNG wire#w11
      R_Coil( "62" )
   END_RUNG
   RUNG wire#w11
      R_Coil( "63" )
   END_RUNG
   RUNG wire#powerrail
      Contact( "65" )
      wire#w12
      R_Coil( "Z" )
   END_RUNG
   RUNG wire#w12
      R_Coil( "LA" )
   END_RUNG
   RUNG wire#w12
      R_Coil( "LD" )
   END_RUNG
   RUNG wire#w12
      Coil( "deleteAllCalls" )
   END_RUNG
   RUNG wire#w12
      R_Coil( "65" )
   END_RUNG
   RUNG wire#powerrail
      Contact( "62" )
      wire#w13
      Contact( "BD" )
      wire#w14
      S_Coil( "66" )
   END_RUNG
   RUNG wire#powerrail
      Contact( "63" )
   END_RUNG wire#w13
   RUNG wire#w14
      R_Coil( "62" )
   END_RUNG
   RUNG wire#w14
      R_Coil( "63" )
   END_RUNG
   RUNG wire#powerrail
      Contact( "66" )
      wire#w15
      R_Coil( "Z" )
   END_RUNG
   RUNG wire#w15
      R_Coil( "LD" )
   END_RUNG
   RUNG wire#w15
      S_Coil( "moveDown" )
   END_RUNG
   RUNG wire#w15
      R_Coil( "66" )
   END_RUNG
   // the same network as SCL:
   IF NOT "modoSeguridad" AND "sistemaActivado" AND "modoManual" AND "esperandoOrden" THEN
       "60" := TRUE;
   END_IF;
   IF "60" AND "upCall" AND NOT "downCall" THEN
       "61" := TRUE;
       "60" := FALSE;
   END_IF;
   IF "61" THEN
       "Z" := TRUE;
       "LA" := TRUE;
   END_IF;
   IF "60" AND "upCall" AND "downCall" THEN
       "62" := TRUE;
       "60" := FALSE;
   END_IF;
   IF "62" THEN
       "Z" := TRUE;
       "LA" := TRUE;
       "LD" := TRUE;
   END_IF;
   IF "60" AND NOT "upCall" AND "downCall" THEN
       "63" := TRUE;
       "60" := FALSE;
   END_IF;
   IF "63" THEN
       "Z" := TRUE;
       "LD" := TRUE;
   END_IF;
   IF ("61" OR "62") AND "BA" THEN "64" := TRUE; END_IF;
   #_w1 := ("61" OR "62") AND "BA";
   IF #_w1 THEN
       "61" := FALSE;
       "62" := FALSE;
   END_IF;
   IF "64" THEN
       "Z" := FALSE;
       "LA" := FALSE;
       "moveUp" := TRUE;
       "64" := FALSE;
   END_IF;
   IF ("61" OR "62" OR "63") AND "BI" THEN "65" := TRUE; END_IF;
   #_w2 := ("61" OR "62" OR "63") AND "BI";
   IF #_w2 THEN
       "61" := FALSE;
       "62" := FALSE;
       "63" := FALSE;
   END_IF;
   IF "65" THEN
       "Z" := FALSE;
       "LA" := FALSE;
       "LD" := FALSE;
   END_IF;
   "deleteAllCalls" := "65";
   IF "65" THEN "65" := FALSE; END_IF;
   IF ("62" OR "63") AND "BD" THEN "66" := TRUE; END_IF;
   #_w3 := ("62" OR "63") AND "BD";
   IF #_w3 THEN
       "62" := FALSE;
       "63" := FALSE;
   END_IF;
   IF "66" THEN
       "Z" := FALSE;
       "LD" := FALSE;
       "moveDown" := TRUE;
       "66" := FALSE;
   END_IF;
END_REGION

REGION Network 13: Detección de errores
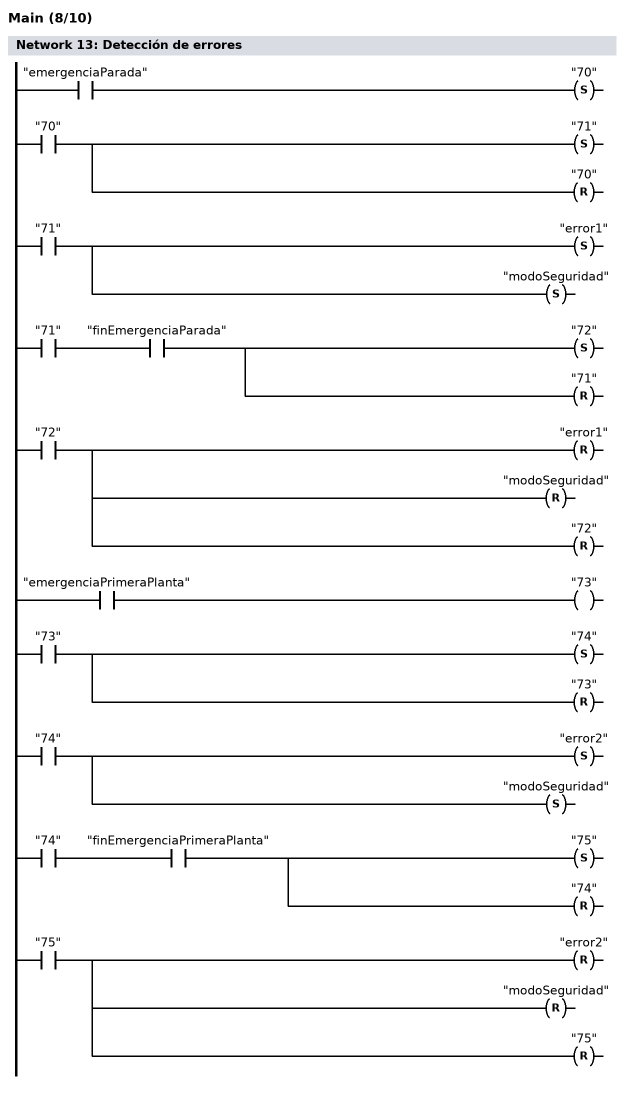
   RUNG wire#powerrail
      Contact( "emergenciaParada" )
      S_Coil( "70" )
   END_RUNG
   RUNG wire#powerrail
      Contact( "70" )
      wire#w1
      S_Coil( "71" )
   END_RUNG
   RUNG wire#w1
      R_Coil( "70" )
   END_RUNG
   RUNG wire#powerrail
      Contact( "71" )
      wire#w2
      S_Coil( "error1" )
   END_RUNG
   RUNG wire#w2
      S_Coil( "modoSeguridad" )
   END_RUNG
   RUNG wire#powerrail
      Contact( "71" )
      Contact( "finEmergenciaParada" )
      wire#w3
      S_Coil( "72" )
   END_RUNG
   RUNG wire#w3
      R_Coil( "71" )
   END_RUNG
   RUNG wire#powerrail
      Contact( "72" )
      wire#w4
      R_Coil( "error1" )
   END_RUNG
   RUNG wire#w4
      R_Coil( "modoSeguridad" )
   END_RUNG
   RUNG wire#w4
      R_Coil( "72" )
   END_RUNG
   RUNG wire#powerrail
      Contact( "emergenciaPrimeraPlanta" )
      Coil( "73" )
   END_RUNG
   RUNG wire#powerrail
      Contact( "73" )
      wire#w5
      S_Coil( "74" )
   END_RUNG
   RUNG wire#w5
      R_Coil( "73" )
   END_RUNG
   RUNG wire#powerrail
      Contact( "74" )
      wire#w6
      S_Coil( "error2" )
   END_RUNG
   RUNG wire#w6
      S_Coil( "modoSeguridad" )
   END_RUNG
   RUNG wire#powerrail
      Contact( "74" )
      Contact( "finEmergenciaPrimeraPlanta" )
      wire#w7
      S_Coil( "75" )
   END_RUNG
   RUNG wire#w7
      R_Coil( "74" )
   END_RUNG
   RUNG wire#powerrail
      Contact( "75" )
      wire#w8
      R_Coil( "error2" )
   END_RUNG
   RUNG wire#w8
      R_Coil( "modoSeguridad" )
   END_RUNG
   RUNG wire#w8
      R_Coil( "75" )
   END_RUNG
   // the same network as SCL:
   IF "emergenciaParada" THEN "70" := TRUE; END_IF;
   IF "70" THEN
       "71" := TRUE;
       "70" := FALSE;
   END_IF;
   IF "71" THEN
       "error1" := TRUE;
       "modoSeguridad" := TRUE;
   END_IF;
   IF "71" AND "finEmergenciaParada" THEN
       "72" := TRUE;
       "71" := FALSE;
   END_IF;
   IF "72" THEN
       "error1" := FALSE;
       "modoSeguridad" := FALSE;
       "72" := FALSE;
   END_IF;
   "73" := "emergenciaPrimeraPlanta";
   IF "73" THEN
       "74" := TRUE;
       "73" := FALSE;
   END_IF;
   IF "74" THEN
       "error2" := TRUE;
       "modoSeguridad" := TRUE;
   END_IF;
   IF "74" AND "finEmergenciaPrimeraPlanta" THEN
       "75" := TRUE;
       "74" := FALSE;
   END_IF;
   IF "75" THEN
       "error2" := FALSE;
       "modoSeguridad" := FALSE;
       "75" := FALSE;
   END_IF;
END_REGION

REGION Network 14: Gestión de errores
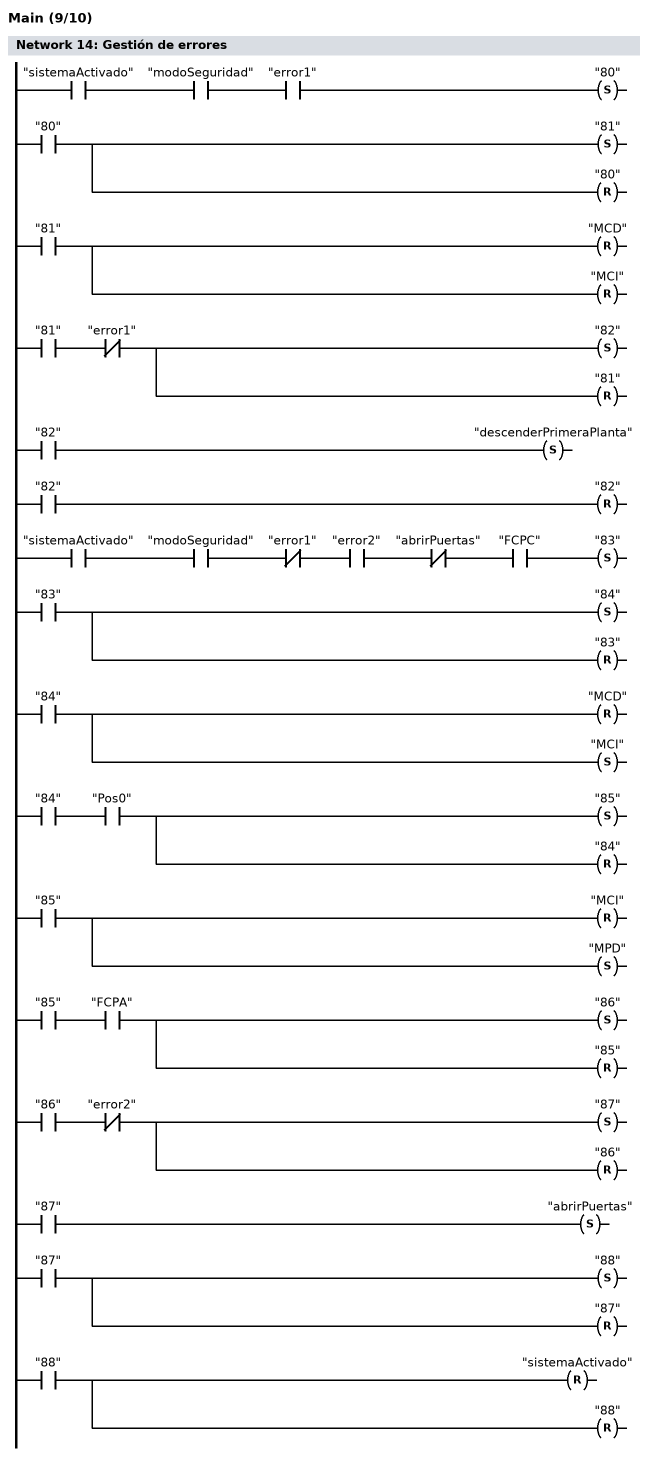
   RUNG wire#powerrail
      Contact( "sistemaActivado" )
      Contact( "modoSeguridad" )
      Contact( "error1" )
      S_Coil( "80" )
   END_RUNG
   RUNG wire#powerrail
      Contact( "80" )
      wire#w1
      S_Coil( "81" )
   END_RUNG
   RUNG wire#w1
      R_Coil( "80" )
   END_RUNG
   RUNG wire#powerrail
      Contact( "81" )
      wire#w2
      R_Coil( "MCD" )
   END_RUNG
   RUNG wire#w2
      R_Coil( "MCI" )
   END_RUNG
   RUNG wire#powerrail
      Contact( "81" )
      I_Contact( "error1" )
      wire#w3
      S_Coil( "82" )
   END_RUNG
   RUNG wire#w3
      R_Coil( "81" )
   END_RUNG
   RUNG wire#powerrail
      Contact( "82" )
      S_Coil( "descenderPrimeraPlanta" )
   END_RUNG
   RUNG wire#powerrail
      Contact( "82" )
      R_Coil( "82" )
   END_RUNG
   RUNG wire#powerrail
      Contact( "sistemaActivado" )
      Contact( "modoSeguridad" )
      I_Contact( "error1" )
      Contact( "error2" )
      I_Contact( "abrirPuertas" )
      Contact( "FCPC" )
      S_Coil( "83" )
   END_RUNG
   RUNG wire#powerrail
      Contact( "83" )
      wire#w4
      S_Coil( "84" )
   END_RUNG
   RUNG wire#w4
      R_Coil( "83" )
   END_RUNG
   RUNG wire#powerrail
      Contact( "84" )
      wire#w5
      R_Coil( "MCD" )
   END_RUNG
   RUNG wire#w5
      S_Coil( "MCI" )
   END_RUNG
   RUNG wire#powerrail
      Contact( "84" )
      Contact( "Pos0" )
      wire#w6
      S_Coil( "85" )
   END_RUNG
   RUNG wire#w6
      R_Coil( "84" )
   END_RUNG
   RUNG wire#powerrail
      Contact( "85" )
      wire#w7
      R_Coil( "MCI" )
   END_RUNG
   RUNG wire#w7
      S_Coil( "MPD" )
   END_RUNG
   RUNG wire#powerrail
      Contact( "85" )
      Contact( "FCPA" )
      wire#w8
      S_Coil( "86" )
   END_RUNG
   RUNG wire#w8
      R_Coil( "85" )
   END_RUNG
   RUNG wire#powerrail
      Contact( "86" )
      I_Contact( "error2" )
      wire#w9
      S_Coil( "87" )
   END_RUNG
   RUNG wire#w9
      R_Coil( "86" )
   END_RUNG
   RUNG wire#powerrail
      Contact( "87" )
      S_Coil( "abrirPuertas" )
   END_RUNG
   RUNG wire#powerrail
      Contact( "87" )
      wire#w10
      S_Coil( "88" )
   END_RUNG
   RUNG wire#w10
      R_Coil( "87" )
   END_RUNG
   RUNG wire#powerrail
      Contact( "88" )
      wire#w11
      R_Coil( "sistemaActivado" )
   END_RUNG
   RUNG wire#w11
      R_Coil( "88" )
   END_RUNG
   // the same network as SCL:
   IF "sistemaActivado" AND "modoSeguridad" AND "error1" THEN "80" := TRUE; END_IF;
   IF "80" THEN
       "81" := TRUE;
       "80" := FALSE;
   END_IF;
   IF "81" THEN
       "MCD" := FALSE;
       "MCI" := FALSE;
   END_IF;
   IF "81" AND NOT "error1" THEN
       "82" := TRUE;
       "81" := FALSE;
   END_IF;
   IF "82" THEN
       "descenderPrimeraPlanta" := TRUE;
       "82" := FALSE;
   END_IF;
   IF "sistemaActivado" AND "modoSeguridad" AND NOT "error1" AND "error2" AND NOT "abrirPuertas" AND "FCPC" THEN
       "83" := TRUE;
   END_IF;
   IF "83" THEN
       "84" := TRUE;
       "83" := FALSE;
   END_IF;
   IF "84" THEN
       "MCD" := FALSE;
       "MCI" := TRUE;
   END_IF;
   IF "84" AND "Pos0" THEN
       "85" := TRUE;
       "84" := FALSE;
   END_IF;
   IF "85" THEN
       "MCI" := FALSE;
       "MPD" := TRUE;
   END_IF;
   IF "85" AND "FCPA" THEN
       "86" := TRUE;
       "85" := FALSE;
   END_IF;
   IF "86" AND NOT "error2" THEN
       "87" := TRUE;
       "86" := FALSE;
   END_IF;
   IF "87" THEN
       "abrirPuertas" := TRUE;
       "88" := TRUE;
       "87" := FALSE;
   END_IF;
   IF "88" THEN
       "sistemaActivado" := FALSE;
       "88" := FALSE;
   END_IF;
END_REGION

REGION Network 15: Descenso a Primera Planta
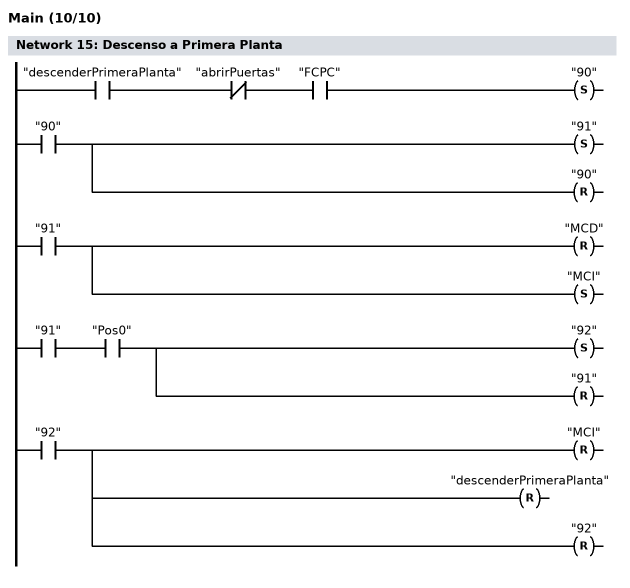
   RUNG wire#powerrail
      Contact( "descenderPrimeraPlanta" )
      I_Contact( "abrirPuertas" )
      Contact( "FCPC" )
      S_Coil( "90" )
   END_RUNG
   RUNG wire#powerrail
      Contact( "90" )
      wire#w1
      S_Coil( "91" )
   END_RUNG
   RUNG wire#w1
      R_Coil( "90" )
   END_RUNG
   RUNG wire#powerrail
      Contact( "91" )
      wire#w2
      R_Coil( "MCD" )
   END_RUNG
   RUNG wire#w2
      S_Coil( "MCI" )
   END_RUNG
   RUNG wire#powerrail
      Contact( "91" )
      Contact( "Pos0" )
      wire#w3
      S_Coil( "92" )
   END_RUNG
   RUNG wire#w3
      R_Coil( "91" )
   END_RUNG
   RUNG wire#powerrail
      Contact( "92" )
      wire#w4
      R_Coil( "MCI" )
   END_RUNG
   RUNG wire#w4
      R_Coil( "descenderPrimeraPlanta" )
   END_RUNG
   RUNG wire#w4
      R_Coil( "92" )
   END_RUNG
   // the same network as SCL:
   IF "descenderPrimeraPlanta" AND NOT "abrirPuertas" AND "FCPC" THEN "90" := TRUE; END_IF;
   IF "90" THEN
       "91" := TRUE;
       "90" := FALSE;
   END_IF;
   IF "91" THEN
       "MCD" := FALSE;
       "MCI" := TRUE;
   END_IF;
   IF "91" AND "Pos0" THEN
       "92" := TRUE;
       "91" := FALSE;
   END_IF;
   IF "92" THEN
       "MCI" := FALSE;
       "descenderPrimeraPlanta" := FALSE;
       "92" := FALSE;
   END_IF;
END_REGION
END_ORGANIZATION_BLOCK